// TIA Portal V20 export
TYPE "LConSMC_typeOperationDynamics"
// [Einheit der Achse] Dynamiken die im Normalbetrieb wirken (müssen größer oder gleich denen des Leitwertes sein!!)  Wirksam wenn "enable" & "speedMatch" & "ctrlEnable" = TRUE / [Unit of the axis] Dynamics during normal operation  Active if "enable" & "speedMatch" & "ctrlEnable" = TRUE
// stored: Access Published
   STRUCT
      acceleration : Real := -1.0;   // Beschleunigung in Achseinheit / Acceleration value: Units are taken from the TO
      deceleration : Real := -1.0;   // Verzögerung in Achseinheit / Deceleration value: Units are taken from the TO
      jerk : Real := -1.0;   // Ruckbegrenzung in Achseinheit / Jerk value : Units are taken from the TO
   END_STRUCT;
END_TYPE
